TEXTLIST CRAH_Status
  0 = 'Hand'
  1 = 'Off'
  2 = 'Auto'
   = ''
END_TEXTLIST

(* stored: Version 1.1.0.1, ProductVersion 3.1.4024.12
   TextList CRAH_Status: Id {2efd7530-e9c7-4963-bde8-1b420f5b2445} *)
